// TIA Portal project "HowCreateTask_" (V16)

(* hardware
DEVICE "ET 200SP station_1"  ET 200SP-Station
   slot 0: "Rack_0"  Rack  6ES5 710-8MAx1
   slot 1: "PLC_1"  CPU 1510SP-1 PN  6ES7 510-1DJ00-0AB0  V1.8
      slot 32768: "PROFINET interface_1"  X1
         slot 32771: "Port_3"  X1 P3
   slot 2: "Server module_1"  Server module  6ES7 193-6PA00-0AA0  V1.1
      slot 1: "Server module_1"  Server module
   slot 127: "BA 2xRJ45"  BA 2xRJ45  6ES7 193-6AR00-0AA0  V0.0
      slot 32769: "Port_1"  X1 P1  6ES7 193-6AR00-0AA0
      slot 32770: "Port_2"  X1 P2  6ES7 193-6AR00-0AA0
*)

// ===== PLC "PLC_1"  CPU 1510SP-1 PN =====

TYPE "tyConcatorTask"
   STRUCT
      Inputs : Struct
         InputReq : Bool;
      END_STRUCT;
      OutputsStates : Struct
         Ready : Bool;
         Busy : Bool;
         Done : Bool;
      END_STRUCT;
   END_STRUCT;
END_TYPE

// folder: ContactorDataType

TYPE "tyContactor_Input"
   STRUCT
      bContactorStartRequest : Bool;
      bContactorFeedbackInput : Bool;
   END_STRUCT;
END_TYPE

TYPE "tyContactor_Output"
   STRUCT
      bActivateContactorCoil : Bool;
      bContactorFault : Bool;
      b_MotorIsRunning : Bool;
   END_STRUCT;
END_TYPE

TYPE "tyContactor_StaticData"
   STRUCT
      TContactorControllTimer : TON_TIME;
      TcontactorFeedBackControlTime : Time;
   END_STRUCT;
END_TYPE

TYPE "tyContactor_Main"
   STRUCT
      ContactorInputs : "tyContactor_Input";
      ContactorOutputs : "tyContactor_Output";
      ContactorStatic : "tyContactor_StaticData";
   END_STRUCT;
END_TYPE

// folder: (top level)

DATA_BLOCK "tContactorControlTask_DB"   // DB1
{ S7_Optimized_Access := 'TRUE' }
VERSION : 0.1
// stored: InstanceOfName tContactorControlTask
"tContactorControlTask"
BEGIN
END_DATA_BLOCK

FUNCTION_BLOCK "oContactorControll_Obj"   // FB1, SCL
{ S7_Optimized_Access := 'TRUE' }
VERSION : 0.1
   VAR
      MotorContactorControll : Array[0..10] of "tyContactor_Main";
   END_VAR
   VAR_TEMP
      i : Int;
   END_VAR
BEGIN
   //=============================================================================
   // Dmitri Raihtsaum - Copyright 2023
   // Created By: Dmitri Raihtsaum
   //-----------------------------------------------------------------------------
   // Tested with:   CPU 1510SP-1 PN
   // Engineering:   TIA Portal V16
   // Functionality: Contactor Control Object 
   // Date: 09.04.2023
   // Rev 0.1
   //=============================================================================

   FOR #i := 0 TO 10 DO

       //Mapping
       #MotorContactorControll[#i].ContactorStatic.TcontactorFeedBackControlTime := t#2s;
       //Logic
       //Contactor Start signal 
       IF #MotorContactorControll[#i].ContactorInputs.bContactorStartRequest THEN
           #MotorContactorControll[#i].ContactorOutputs.bActivateContactorCoil := TRUE;
       END_IF;
       //Contactor Stop signal
       IF NOT #MotorContactorControll[#i].ContactorInputs.bContactorStartRequest THEN
           #MotorContactorControll[#i].ContactorOutputs.bActivateContactorCoil := FALSE;
       END_IF;
       //Check Contactor Status 
       IF #MotorContactorControll[#i].ContactorOutputs.bActivateContactorCoil THEN 
           //AND #MotorContactorControll[#i].ContactorInputs.bContactorFeedbackInput THEN
           #MotorContactorControll[#i].ContactorOutputs.b_MotorIsRunning := TRUE;
       ELSE
           #MotorContactorControll[#i].ContactorOutputs.b_MotorIsRunning := FALSE;
       END_IF;
       // Fault Signal
     //  IF #MotorContactorControll[#i].ContactorInputs.bContactorStartRequest AND NOT #MotorContactorControll[#i].ContactorInputs.bContactorFeedbackInput
     //      OR NOT #MotorContactorControll[#i].ContactorInputs.bContactorStartRequest AND #MotorContactorControll[#i].ContactorInputs.bContactorFeedbackInput
    //   THEN
     //      #MotorContactorControll[#i].ContactorStatic.TContactorControllTimer(IN := TRUE,
       //                                                                        PT := #MotorContactorControll[#i].ContactorStatic.TcontactorFeedBackControlTime);
     //  ELSE
     //      #MotorContactorControll[#i].ContactorStatic.TContactorControllTimer(IN := FALSE,
     //                                                                          PT := t#0ms);
     //  END_IF;
       // Fault Flag
       IF #MotorContactorControll[#i].ContactorStatic.TContactorControllTimer.Q THEN
           #MotorContactorControll[#i].ContactorOutputs.bContactorFault := TRUE;
       ELSE
           #MotorContactorControll[#i].ContactorOutputs.bContactorFault := FALSE;
       END_IF;
   END_FOR;
   //=============================================================================
   //END
   //=============================================================================
END_FUNCTION_BLOCK

FUNCTION_BLOCK "tContactorControlTask"   // FB2, SCL
{ S7_Optimized_Access := 'TRUE' }
VERSION : 0.1
   VAR
      currentStep : Int;
      Interface : "tyConcatorTask";
      oContactorControll_Obj_Instance : "oContactorControll_Obj";
      StepTimer_0 : TON_TIME;
      StepTimer_1 : TON_TIME;
      StepTimer_2 : TON_TIME;
   END_VAR
   VAR_TEMP
      i : Int;
   END_VAR
BEGIN
   //=============================================================================
   // Dmitri Raihtsaum - Copyright 2023
   // Created By: Dmitri Raihtsaum
   //-----------------------------------------------------------------------------
   // Tested with:   CPU 1510SP-1 PN
   // Engineering:   TIA Portal V16
   // Functionality: Contactor Control Task
   // Date: 21.04.2023
   // Rev 0.1
   //=============================================================================


   CASE #currentStep OF
       0:  // init
           #StepTimer_0(IN := FALSE,
                        PT := t#2s);
           #StepTimer_1(IN := FALSE,
                        PT := t#2s);
           #StepTimer_2(IN := FALSE,
                        PT := t#2s);
           #Interface.OutputsStates.Ready := TRUE;
           #Interface.OutputsStates.Busy := FALSE;
           #Interface.OutputsStates.Done := FALSE;
           FOR #i := 0 TO 10 DO
               #oContactorControll_Obj_Instance.MotorContactorControll[#i].ContactorInputs.bContactorStartRequest := FALSE;
           END_FOR;
           IF #Interface.Inputs.InputReq THEN
               #currentStep := 1;
           END_IF;

       1:  // Start motor (0)
           #Interface.OutputsStates.Ready := FALSE;
           #Interface.OutputsStates.Busy := TRUE;
           #Interface.OutputsStates.Done := FALSE;
           #oContactorControll_Obj_Instance.MotorContactorControll[0].ContactorInputs.bContactorStartRequest := TRUE;
           IF #oContactorControll_Obj_Instance.MotorContactorControll[0].ContactorOutputs.b_MotorIsRunning THEN
               #StepTimer_0(IN := TRUE,
                            PT := t#2s);
               IF #StepTimer_0.Q THEN
                   #currentStep := 2;
               END_IF;
           END_IF;

       2: // Start motor (1)
           #oContactorControll_Obj_Instance.MotorContactorControll[1].ContactorInputs.bContactorStartRequest := TRUE;
           IF #oContactorControll_Obj_Instance.MotorContactorControll[1].ContactorOutputs.b_MotorIsRunning THEN
               #StepTimer_1(IN := TRUE,
                            PT := t#2s);
               IF #StepTimer_1.Q THEN
                   #currentStep := 3;
               END_IF;
           END_IF;
           ;
       3:  // Start motor (2)
           #oContactorControll_Obj_Instance.MotorContactorControll[2].ContactorInputs.bContactorStartRequest := TRUE;
           IF #oContactorControll_Obj_Instance.MotorContactorControll[2].ContactorOutputs.b_MotorIsRunning THEN
               #StepTimer_2(IN := TRUE,
                            PT := t#2s);
               IF #StepTimer_2.Q THEN
                   #currentStep := 4;
               END_IF;
           END_IF;

       4: //Task Done - Stop  all motors
           #Interface.OutputsStates.Ready := FALSE;
           #Interface.OutputsStates.Busy := FALSE;
           #Interface.OutputsStates.Done := TRUE;
           FOR #i := 0 TO 10 DO
               #oContactorControll_Obj_Instance.MotorContactorControll[#i].ContactorInputs.bContactorStartRequest := FALSE;
           END_FOR;

   END_CASE;
   IF NOT #Interface.Inputs.InputReq THEN
       #currentStep := 0;
   END_IF;

   #oContactorControll_Obj_Instance();
END_FUNCTION_BLOCK

ORGANIZATION_BLOCK "Main"   // OB1, LAD, ProgramCycle
TITLE = "Main Program Sweep (Cycle)"
{ S7_Optimized_Access := 'TRUE' }
VERSION : 0.1
   VAR_INPUT
      Initial_Call : Bool;   // Initial call of this OB
      Remanence : Bool;   // =True, if remanent data are available
   END_VAR
BEGIN

REGION Network 2
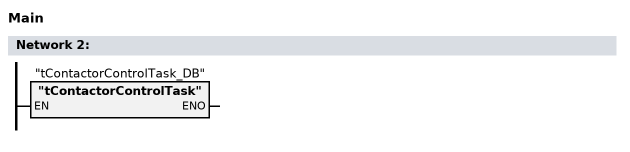
   RUNG wire#powerrail
      "tContactorControlTask_DB"()
   END_RUNG
   // the same network as SCL:
   "tContactorControlTask_DB"();   // "tContactorControlTask"
END_REGION
END_ORGANIZATION_BLOCK